{attribute 'qualified_only'}
VAR_GLOBAL CONSTANT
	// Encoder reference values in counts = nm
	// Enc Ref Vals from alignment 2020-6-12
	nYUP_ENC_REF : ULINT := 14279350;
	nYDWN_ENC_REF : ULINT := 15196760;
	nXUP_ENC_REF : ULINT := 25135760;
	nXDWN_ENC_REF : ULINT := 24091270;
END_VAR

(* stored: Version 1.1.0.1, ProductVersion 3.1.4022.18
   GVL GVL_MR2L3_Constants: Id {a89c8f55-2337-47fa-9d19-39ce2e9d821e} *)
